// TIA Portal project "Lab6" (V16)

(* hardware
DEVICE "S71500/ET200MP station_1"  S7-1500 station
   slot 0: "Perfil soporte_0"  Rack  6ES7 590-1***0-0AA0
   slot 0: "PM 70W 120/230VAC"  PM 70W 120/230VAC  6EP1332-4BA00
   slot 1: "PLC_1"  CPU 1512C-1 PN  6ES7 512-1CK00-0AB0  V1.8
      slot 3: "Display de la CPU_1"  6ES7591-1AA00-0AA0
      slot 32768: "Interfaz PROFINET_1"  X1
   slot 2: "CP 1542-5_1"  CP 1542-5  6GK7 542-5FX00-0XE0  V1.0
DEVICE "PC-System_1"  SIMATIC PC station
   slot 0: "Estación PC SIMATIC"  Rail  SIMATIC PC-Station  V1.0
      slot 125: "Stationmanager"  Station_Manager  V6.0.4
   slot 1: "HMI_RT_1"  WinCC RT Advanced  6AV2 104-0xxxx-xxxx  16.0.0.0
      slot 33792: "Interfaz del equipo"  Host interface
   slot 2: "IE general_1"  IE General  IE_CP  V8.2.0
DEVICE "HMI_1"  KTP700 Basic PN
   slot 0: "HMI_1"  KTP700 Basic PN  6AV2 123-2GB03-0AX0  16.0.0.0
   slot 1: "HMI_RT_2"  KTP700 Basic PN  6AV2 123-2GB03-0AX0  16.0.0.0
   slot 5: "HMI_1.IE_CP_1"  PROFINET Interface  16.0.0.0
      slot 1: "Interfaz PROFINET_1"  PROFINET Interface
         slot 1: "Port_1"  Port
DEVICE "SINAMICS G_1"  Sinamics.Device
   slot 0: "	_0"  Rail  SinamicsG120SVecto
   slot 0: "accionamiento_1"  G120 CU250S-2 PN Vector  6SL3246-0BA22-1FA0  4.7.6
      slot 1: "Interfaz PROFINET"  MDD-SinamicsG120-P
   slot 3: "PM240-2 IP20"  PM240-2 IP20  6SL3210-1PB13-8ULx  -
DEVICE "S71500/ET200MP station_2"  S7-1500 station
   slot 0: "Perfil soporte_0"  Rack  6ES7 590-1***0-0AA0
   slot 1: "PLC_2"  CPU 1512C-1 PN  6ES7 512-1CK00-0AB0  V1.8
      slot 3: "Display de la CPU_1"  6ES7591-1AA00-0AA0
      slot 32768: "Interfaz PROFINET_1"  X1
   slot 2: "CP 1542-5_1"  CP 1542-5  6GK7 542-5FX00-0XE0  V1.0
*)

// ===== PLC "PLC_1"  CPU 1512C-1 PN =====

VAR_GLOBAL   // PLC tag table "Tabla de variables estándar"
   "Referencia(°C)" AT %MD14 : Real;
   "PT100" AT %IW20 : Int;
   "Bombillo" AT %Q4.7 : Bool;
   "Temperatura_Normal" AT %MD0 : Real;
   "Temperatura_Medida" AT %MD4 : Real;
   "Star" AT %M10.0 : Bool;
   "Stop" AT %M20.1 : Bool;
   "Paro" AT %M100.2 : Bool;
   "Servomotor" AT %Q16.1 : Bool;
   "Error" AT %MD104 : Real;
   "Alarma_Referencia_Alcanzada" AT %Q0.2 : Bool;
   "Encender_Variador" AT %M12.0 : Bool;
   "Stop_fisico" AT %I30.2 : Bool;
   "Parofisico" AT %I30.3 : Bool;
   "Star_Fisico" AT %I30.1 : Bool;
   "MoverDerecha" AT %M10.3 : Bool;
   "Pid_Sintonizado" AT %M8.0 : Bool;
   "Alarma_Alta" AT %Q16.3 : Bool;
   "Alarma_Baja" AT %Q16.4 : Bool;
   "Variador" AT %Q16.7 : Bool;
   "Ventilador" AT %Q16.6 : Bool;
   "Pid_Manual" AT %M8.1 : Bool;
   "Servosistema" AT %M8.2 : Bool;
   "Pid_Discreto" AT %M8.3 : Bool;
   "Control_Discreto" AT %MD22 : Real;
   "Control_Servo" AT %MD26 : Real;
   "Control_Servo(1)" AT %MD30 : Real;
   "Tag_1" AT %Q16.5 : Bool;
   "Error_Temperatura" AT %MD34 : Real;
END_VAR

DATA_BLOCK "Bloque_1_DB"   // DB4
{ S7_Optimized_Access := 'TRUE' }
VERSION : 0.1
// stored: InstanceOfName Bloque_1
"Bloque_1"
BEGIN
END_DATA_BLOCK

DATA_BLOCK "Base_de_Datos"   // DB5
{ S7_Optimized_Access := 'TRUE' }
VERSION : 0.1
BEGIN
END_DATA_BLOCK

// folder: System blocks/Program resources

DATA_BLOCK "IEC_Timer_0_DB"   // DB2
{ S7_Optimized_Access := 'TRUE' }
AUTHOR : Simatic
FAMILY : IEC
NAME : IEC_TMR
VERSION : 1.0
// stored: InstanceOfName IEC_TIMER
"IEC_TIMER"
BEGIN
END_DATA_BLOCK

DATA_BLOCK "IEC_Timer_0_DB_1"   // DB6
{ S7_Optimized_Access := 'TRUE' }
AUTHOR : Simatic
FAMILY : IEC
NAME : IEC_TMR
VERSION : 1.0
// stored: InstanceOfName IEC_TIMER
"IEC_TIMER"
BEGIN
END_DATA_BLOCK

DATA_BLOCK "IEC_Timer_0_DB_2"   // DB7
{ S7_Optimized_Access := 'TRUE' }
AUTHOR : Simatic
FAMILY : IEC
NAME : IEC_TMR
VERSION : 1.0
// stored: InstanceOfName IEC_TIMER
"IEC_TIMER"
BEGIN
END_DATA_BLOCK

// folder: (top level)

DATA_BLOCK "SpeedAxis_1"   // DB3, Motion_DB
{ S7_Optimized_Access := 'TRUE' }
AUTHOR : SIMATIC
FAMILY : MC_1500
VERSION : 2.0
// stored: InstanceOfName TO_SpeedAxis
"TO_SpeedAxis"
BEGIN
   DynamicLimits.MaxAcceleration := 1000.0;
   DynamicLimits.MaxDeceleration := 1000.0;
   DynamicLimits.MaxJerk := 20000.0;
   DynamicDefaults.Acceleration := 200.0;
   DynamicDefaults.Deceleration := 200.0;
   DynamicDefaults.Jerk := 4000.0;
   DynamicDefaults.EmergencyDeceleration := 1000.0;
   Actor.Interface.AddressIn := 256;
   Actor.Interface.AddressOut := 256;
END_DATA_BLOCK

FUNCTION_BLOCK "Bloque_1"   // FB1, FBD
{ S7_Optimized_Access := 'TRUE' }
VERSION : 0.1
   VAR
      MC_POWER_Instance : MC_POWER;
      MC_RESET_Instance : MC_RESET;
      MC_MOVEJOG_Instance : MC_MOVEJOG;
   END_VAR
BEGIN

REGION Network 1
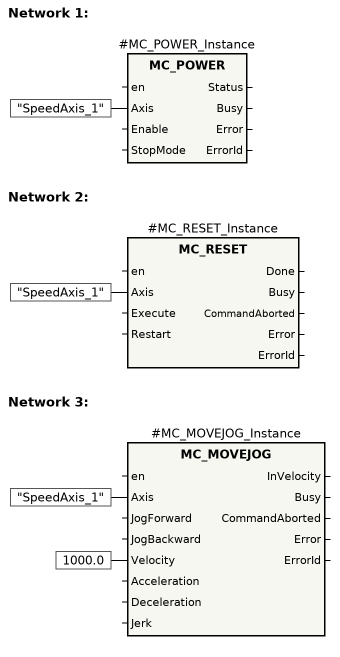
   #MC_POWER_Instance(Axis := "SpeedAxis_1");   // MC_POWER
END_REGION

REGION Network 2
   #MC_RESET_Instance(Axis := "SpeedAxis_1");   // MC_RESET
END_REGION

REGION Network 3
   #MC_MOVEJOG_Instance(Axis := "SpeedAxis_1", Velocity := 1000.0);   // MC_MOVEJOG
END_REGION
END_FUNCTION_BLOCK

ORGANIZATION_BLOCK "Main"   // OB1, LAD, ProgramCycle
TITLE = "Main Program Sweep (Cycle)"
{ S7_Optimized_Access := 'TRUE' }
VERSION : 0.1
   VAR_INPUT
      Initial_Call : Bool;   // Initial call of this OB
      Remanence : Bool;   // =True, if remanent data are available
   END_VAR
   VAR_TEMP
      Encender_Bombillo : Bool;
      Ventilador : Bool;
      calculo_error : Bool;
   END_VAR
BEGIN

REGION Network 1: Normalizar y escalar señal
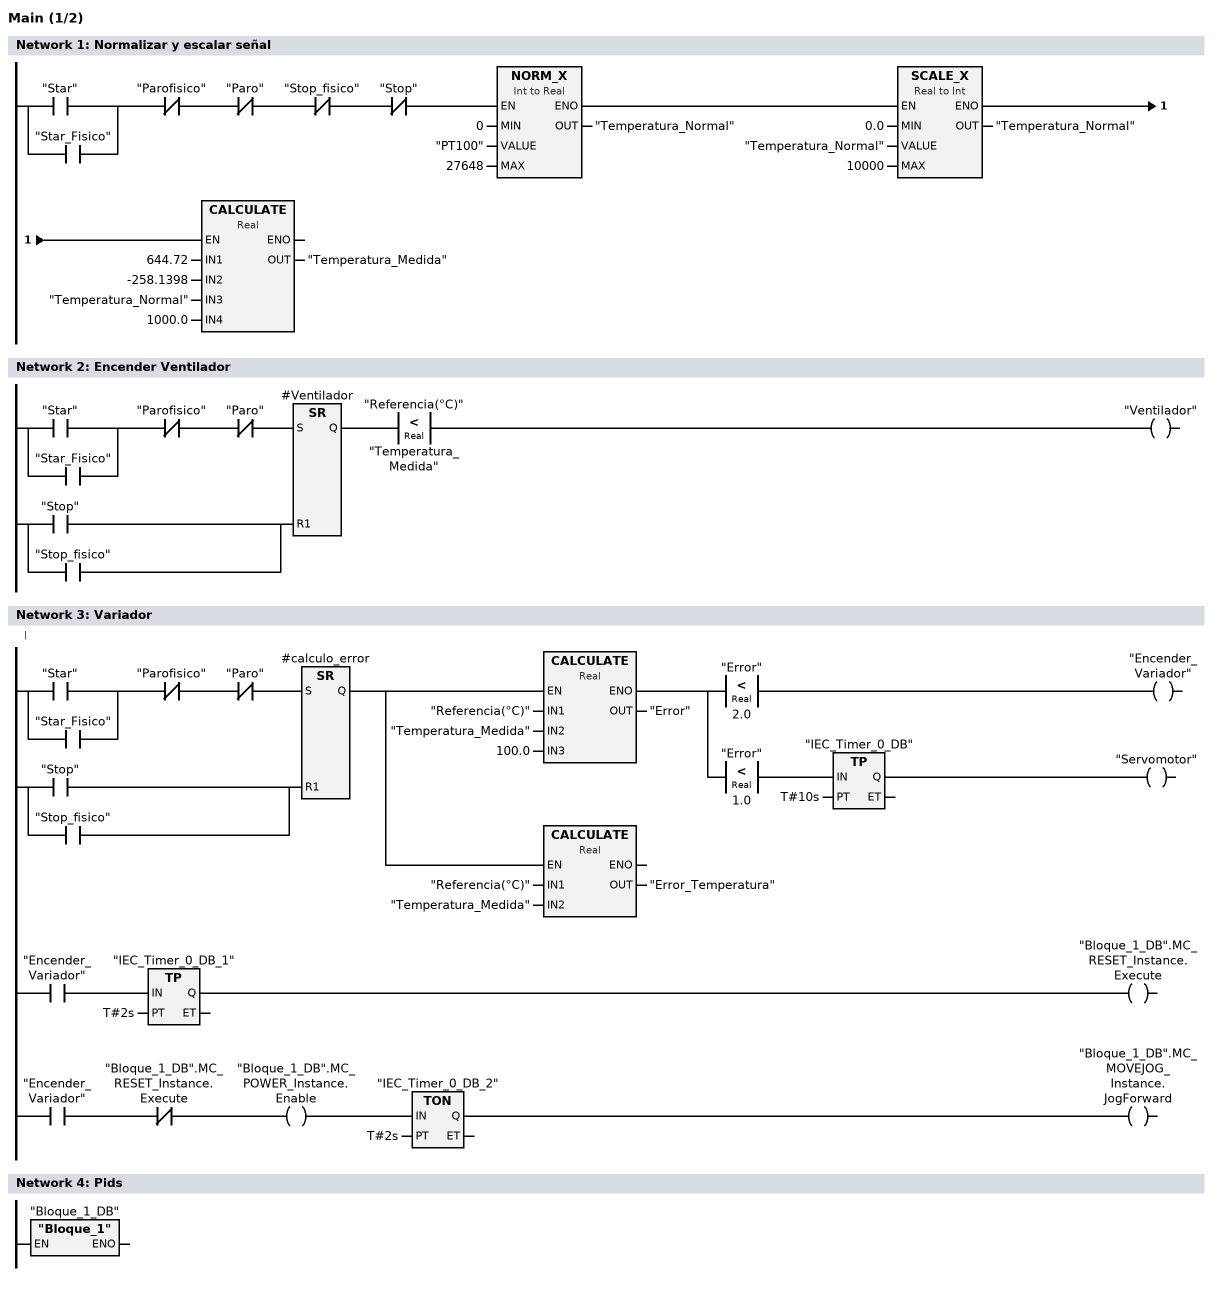
   RUNG wire#powerrail
      Contact( "Star" )
      wire#w1
      I_Contact( "Parofisico" )
      I_Contact( "Paro" )
      I_Contact( "Stop_fisico" )
      I_Contact( "Stop" )
      { S7_Templates := "[SrcType := Int, DestType := Real]" } Normalize(min := 0, value := "PT100", max := 27648, out => "Temperatura_Normal")
      { S7_Templates := "[SrcType := Real, DestType := Int]" } Scale(min := 0.0, value := "Temperatura_Normal", max := 10000, out => "Temperatura_Normal")
      { S7_Templates := "SrcType := Real"; S7_Expression := "(IN1*(IN3/IN4))+IN2" } Calculate(in1 := 644.72, in2 := -258.1398, in3 := "Temperatura_Normal", in4 := 1000.0, out => "Temperatura_Medida")
   END_RUNG
   RUNG wire#powerrail
      Contact( "Star_Fisico" )
   END_RUNG wire#w1
   // the same network as SCL:
   IF ("Star" OR "Star_Fisico") AND NOT "Parofisico" AND NOT "Paro" AND NOT "Stop_fisico" AND NOT "Stop" THEN
       "Temperatura_Normal" := NORM_X(MIN := 0, VALUE := "PT100", MAX := 27648);
       "Temperatura_Normal" := SCALE_X(MIN := 0.0, VALUE := "Temperatura_Normal", MAX := 10000);
       "Temperatura_Medida" := (644.72*("Temperatura_Normal"/1000.0))+(-258.1398);
   END_IF;
END_REGION

REGION Network 2: Encender Ventilador
   RUNG wire#powerrail
      Contact( "Star" )
      wire#w1
      I_Contact( "Parofisico" )
      I_Contact( "Paro" )
      S_SR(operand := #Ventilador, r1 := wire#w2)
      { S7_Templates := "SrcType := Real" } LT_Contact(in1 := "Referencia(°C)", in2 := "Temperatura_Medida")
      Coil( "Ventilador" )
   END_RUNG
   RUNG wire#powerrail
      Contact( "Star_Fisico" )
   END_RUNG wire#w1
   RUNG wire#powerrail
      Contact( "Stop" )
   END_RUNG wire#w2
   RUNG wire#powerrail
      Contact( "Stop_fisico" )
   END_RUNG wire#w2
   // the same network as SCL:
   IF ("Star" OR "Star_Fisico") AND NOT "Parofisico" AND NOT "Paro" THEN
       #Ventilador := TRUE;   // SR flip-flop
   END_IF;
   IF "Stop" OR "Stop_fisico" THEN #Ventilador := FALSE; END_IF;
   "Ventilador" := #Ventilador AND ("Referencia(°C)" < "Temperatura_Medida");
END_REGION

REGION Network 3: Variador
   // l
   IF ("Star" OR "Star_Fisico") AND NOT "Parofisico" AND NOT "Paro" THEN
       #calculo_error := TRUE;   // SR flip-flop
   END_IF;
   IF "Stop" OR "Stop_fisico" THEN #calculo_error := FALSE; END_IF;
   IF #calculo_error THEN
       "Error" := ABS(100.0*("Referencia(°C)"-"Temperatura_Medida")/("Referencia(°C)"));
   END_IF;
   "Encender_Variador" := #calculo_error AND ("Error" < 2.0);
   "IEC_Timer_0_DB".TP(IN := #calculo_error AND ("Error" < 1.0), PT := T#10s);
   "Servomotor" := "IEC_Timer_0_DB".Q;
   IF #calculo_error THEN "Error_Temperatura" := "Referencia(°C)"-"Temperatura_Medida"; END_IF;
   "IEC_Timer_0_DB_1".TP(IN := "Encender_Variador", PT := T#2s);
   "Bloque_1_DB".MC_RESET_Instance.Execute := "IEC_Timer_0_DB_1".Q;
   "Bloque_1_DB".MC_POWER_Instance.Enable := "Encender_Variador" AND NOT "Bloque_1_DB".MC_RESET_Instance.Execute;
   "IEC_Timer_0_DB_2".TON(IN := "Bloque_1_DB".MC_POWER_Instance.Enable, PT := T#2s);
   "Bloque_1_DB".MC_MOVEJOG_Instance.JogForward := "IEC_Timer_0_DB_2".Q;
END_REGION

REGION Network 4: Pids
   RUNG wire#powerrail
      "Bloque_1_DB"()
   END_RUNG
   // the same network as SCL:
   "Bloque_1_DB"();   // "Bloque_1"
END_REGION

REGION Network 5: Alarmas
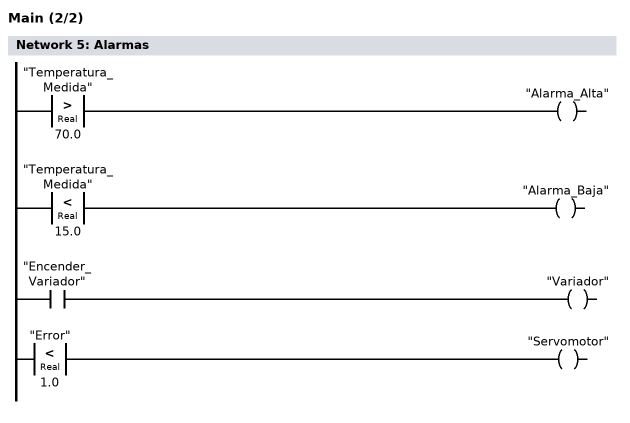
   RUNG wire#powerrail
      { S7_Templates := "SrcType := Real" } GT_Contact(in1 := "Temperatura_Medida", in2 := 70.0)
      Coil( "Alarma_Alta" )
   END_RUNG
   RUNG wire#powerrail
      { S7_Templates := "SrcType := Real" } LT_Contact(in1 := "Temperatura_Medida", in2 := 15.0)
      Coil( "Alarma_Baja" )
   END_RUNG
   RUNG wire#powerrail
      Contact( "Encender_Variador" )
      Coil( "Variador" )
   END_RUNG
   RUNG wire#powerrail
      { S7_Templates := "SrcType := Real" } LT_Contact(in1 := "Error", in2 := 1.0)
      Coil( "Servomotor" )
   END_RUNG
   // the same network as SCL:
   "Alarma_Alta" := "Temperatura_Medida" > 70.0;
   "Alarma_Baja" := "Temperatura_Medida" < 15.0;
   "Variador" := "Encender_Variador";
   "Servomotor" := "Error" < 1.0;
END_REGION
END_ORGANIZATION_BLOCK

ORGANIZATION_BLOCK "Cyclic interrupt_1"   // OB31, LAD, CyclicInterrupt
{ S7_Optimized_Access := 'TRUE' }
VERSION : 0.1
   VAR_INPUT
      Initial_Call : Bool;   // Initial call of this OB
      Event_Count : Int;   // Events discarded
   END_VAR
BEGIN

REGION Network 2: Sintonizado
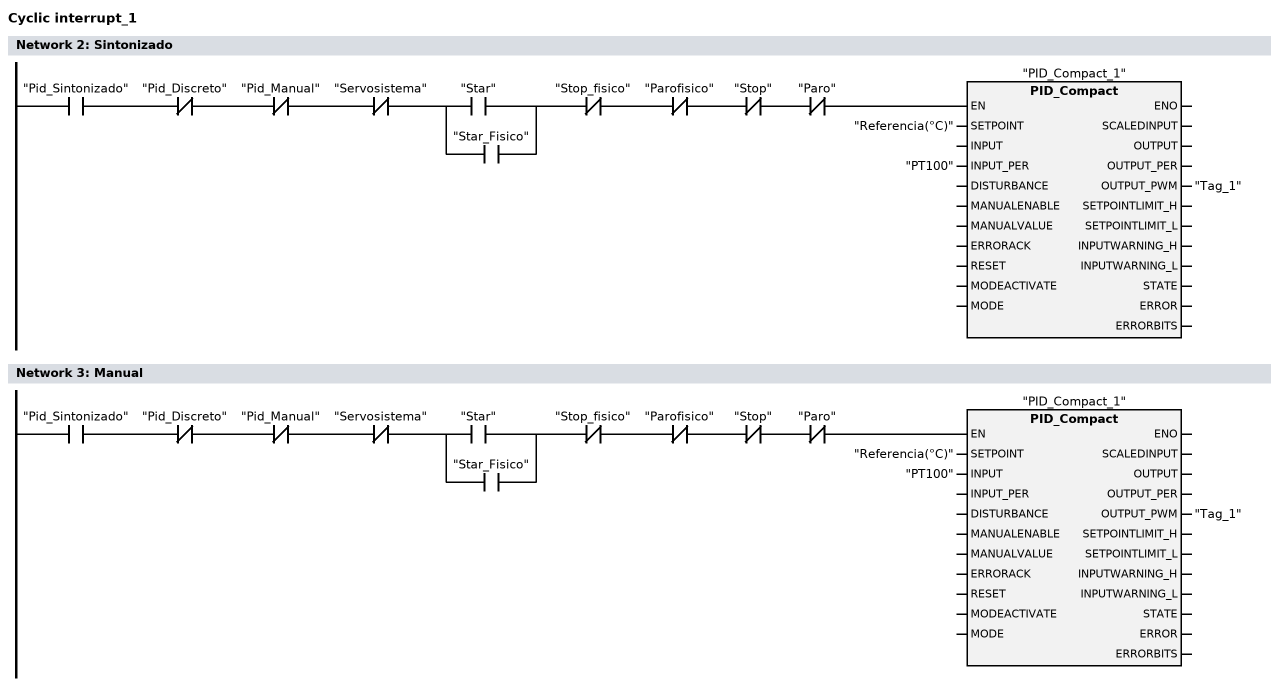
   IF "Pid_Sintonizado" AND NOT "Pid_Discreto" AND NOT "Pid_Manual" AND NOT "Servosistema" AND ("Star" OR "Star_Fisico") AND NOT "Stop_fisico" AND NOT "Parofisico" AND NOT "Stop" AND NOT "Paro" THEN
       "PID_Compact_1"(Setpoint := "Referencia(°C)", Input_PER := "PT100", Output_PWM => "Tag_1");   // PID_Compact
   END_IF;
END_REGION

REGION Network 3: Manual
   IF "Pid_Sintonizado" AND NOT "Pid_Discreto" AND NOT "Pid_Manual" AND NOT "Servosistema" AND ("Star" OR "Star_Fisico") AND NOT "Stop_fisico" AND NOT "Parofisico" AND NOT "Stop" AND NOT "Paro" THEN
       "PID_Compact_1"(Setpoint := "Referencia(°C)", Input := "PT100", Output_PWM => "Tag_1");   // PID_Compact
   END_IF;
END_REGION

REGION Network 4: Servosistema
END_REGION

REGION Network 5: Pid Discreto
END_REGION
END_ORGANIZATION_BLOCK

ORGANIZATION_BLOCK "Main_1"   // OB123, LAD, ProgramCycle
TITLE = "Main Program Sweep (Cycle)"
{ S7_Optimized_Access := 'TRUE' }
VERSION : 0.1
   VAR_INPUT
      Initial_Call : Bool;   // Initial call of this OB
      Remanence : Bool;   // =True, if remanent data are available
   END_VAR
BEGIN
END_ORGANIZATION_BLOCK

// ===== PLC "PLC_2"  CPU 1512C-1 PN =====

ORGANIZATION_BLOCK "Main"   // OB1, LAD, ProgramCycle
TITLE = "Main Program Sweep (Cycle)"
{ S7_Optimized_Access := 'TRUE' }
VERSION : 0.1
   VAR_INPUT
      Initial_Call : Bool;   // Initial call of this OB
      Remanence : Bool;   // =True, if remanent data are available
   END_VAR
BEGIN
END_ORGANIZATION_BLOCK

(* ===== HMI "HMI_RT_1" =====
system functions are stored by id; their names below are inferred from use
connection "HMI_Conexión_1": ETHERNET, S7_1500_OMS
connection "HMI_Conexión_4": ETHERNET, S7_1500_OMS

HMI tags "Tabla de variables estándar"
   "DatabaseName" : WString[254] AT %DB1.DBX0.0
   "ErrDesc" : WString[254], internal
   "TableName" : WString[254] AT %DB1.DBX0.0
   "Column1" : WString[254], internal
   "Column2" : WString[254], internal
   "Column3" : WString[254], internal
   "Referencia(°C)" : Real = PLC "Referencia(°C)" AT %MD14, 1 s
   "PT100" : Int = PLC PT100 AT %IW20, 1 s
   "Bombillo" : Bool = PLC Bombillo AT %Q4.7, 1 s
   "Temperatura_Normal" : Real = PLC Temperatura_Normal AT %MD0, 1 s
   "Temperatura_Medida" : Real = PLC Temperatura_Medida AT %MD4, 1 s
   "Star" : Bool = PLC Star AT %M10.0, 1 s
   "Stop" : Bool = PLC Stop AT %M20.1, 1 s
   "Paro" : Bool = PLC Paro AT %M100.2, 1 s
   "Servomotor" : Bool = PLC Servomotor AT %Q16.1, 1 s
   "Error" : Real = PLC Error AT %MD104, 1 s
   "Alarma_Referencia_Alcanzada" : Bool = PLC Alarma_Referencia_Alcanzada AT %Q0.2, 1 s
   "Encender_Variador" : Bool = PLC Encender_Variador AT %M12.0, 1 s
   "Stop_fisico" : Bool = PLC Stop_fisico AT %I30.2, 1 s
   "Parofisico" : Bool = PLC Parofisico AT %I30.3, 1 s
   "Star_Fisico" : Bool = PLC Star_Fisico AT %I30.1, 1 s
   "MoverDerecha" : Bool = PLC MoverDerecha AT %M10.3, 1 s
   "Pid_Sintonizado" : Bool = PLC Pid_Sintonizado AT %M8.0, 1 s
   "Alarma_Alta" : Bool = PLC Alarma_Alta AT %Q16.3, 1 s
   "Alarma_Baja" : Bool = PLC Alarma_Baja AT %Q16.4, 1 s
   "Variador" : Bool = PLC Variador AT %Q16.7, 1 s
   "Ventilador" : Bool = PLC Ventilador AT %Q16.6, 1 s
   "Pid_Manual" : Bool = PLC Pid_Manual AT %M8.1, 1 s
   "Servosistema" : Bool = PLC Servosistema AT %M8.2, 1 s
   "Pid_Discreto" : Bool = PLC Pid_Discreto AT %M8.3, 1 s
   "Tag_1" : Bool = PLC Tag_1 AT %Q16.5, 1 s
   "Error_Temperatura" : Real = PLC Error_Temperatura AT %MD34, 1 s

screen "Base de Datos" 800x600
   Button "Botón_1" at 22,16 size 209x32; TextOff 'Volver Panel de Control'
      on Press: function_efd93a16()
   IOField "Campo ES_1" at 217,133 size 109x32; FormatPattern 999.99999; Unit °C
      ProcessValue <- "Referencia(°C)"
   IOField "Campo ES_3" at 218,174 size 110x32; FormatPattern 999.99999; Unit °C
      ProcessValue <- "Error"
   TextField "Campo de texto_3" at 163,183 size 40x23; Text 'Error'
   TextField "Campo de texto_2" at 40,142 size 163x23; Text 'Temperatura_Deseada'
   TextField "Campo de texto_4" at 41,101 size 148x23; Text 'Temperatura_Actual'
   IOField "Campo ES_2" at 217,92 size 108x32; FormatPattern 999.99999; Unit °C
      ProcessValue <- "Temperatura_Medida"
   TextField "Campo de texto_1" at 40,62 size 166x23; Text 'Datos Tomados del plc'

screen "Control_Temperatura" 800x600
   Button "Botón_1" at 241,140 size 100x30; TextOff 'Star'
      on Click: SetBit("Star")
   Button "Botón_2" at 241,266 size 100x30; TextOff 'Stop'
      on Click: InvertBit("Stop")
   Button "Botón_3" at 241,202 size 100x30; TextOff 'Paro'
      on Click: InvertBit("Paro")
   IOField "Campo ES_4" at 38,40 size 96x32; FormatPattern 999.99999
      ProcessValue <- "Referencia(°C)"
   TextField "Campo de texto_1" at 7,7 size 209x28; Text 'Temperatura_Deseada'
   Bar "Barra_1" at 390,125 size 141x303; MinimumValue 0; MaximumValue 150
      ProcessValue <- "Temperatura_Medida"
   GraphicView "Visor de gráficos_4" at 25,221 size 161x242; Picture "Gráfico_6"
      Visibility <- "Tag_1"
   GraphicView "Visor de gráficos_3" at 25,221 size 161x242; Picture "Gráfico_7"
      Visibility <- "Tag_1"
   IOField "Campo ES_5" at 56,309 size 98x21; FormatPattern 999.99999
      ProcessValue <- "Temperatura_Medida"
   GraphicView "Visor de gráficos_1" at 162,354 size 95x102; Picture "Gráfico_9"
      Visibility <- "Tag_1"
   GraphicView "Visor de gráficos_2" at 162,354 size 95x102; Picture "Gráfico_9"
      Visibility <- "Tag_1"
   TextField "Campo de texto_4" at 36,163 size 186x28; Text 'Temperatura_Actual'
   Circle "Círculo_1" at 354,9 size 65x65
      Appearance <- "Servomotor"
   Circle "Círculo_2" at 440,8 size 65x65
      Appearance <- "Variador"
   Circle "Círculo_3" at 558,8 size 65x65
      Appearance <- "Alarma_Alta"
   TextField "Campo de texto_5" at 363,72 size 54x28; Text 'Servo'
   TextField "Campo de texto_6" at 437,72 size 79x28; Text 'Variador'
   TextField "Campo de texto_7" at 536,72 size 101x28; Text 'Temp_Alta'
   Circle "Círculo_4" at 680,6 size 65x65
      Appearance <- "Alarma_Baja"
   TextField "Campo de texto_8" at 667,70 size 106x28; Text 'Temp_Baja'
   Button "Botón_4" at 585,187 size 140x30; TextOff 'Pid_Sintonizado'
      on Press: InvertBit("Pid_Sintonizado")
      Appearance <- "Pid_Sintonizado"
   Button "Botón_7" at 30,83 size 140x30; TextOn 'Base de Datos'; TextOff 'Base de Datos'
      on Click: ActivateScreen("Base de Datos", 0)
      on Press: ActivateScreen("Base de Datos", 0)
   Button "Botón_8" at 585,129 size 140x30; TextOff 'Pid_Manual'
      on Press: InvertBit("Pid_Manual")
      Appearance <- "Pid_Manual"
   Button "Botón_9" at 585,237 size 140x30; TextOff 'Servosistema'
      on Press: InvertBit("Servosistema")
      Appearance <- "Servosistema"
   Button "Botón_10" at 585,287 size 140x30; TextOff 'Pid_Discreto'
      on Press: InvertBit("Pid_Discreto")
      Appearance <- "Pid_Discreto"
   Button "Botón_5" at 585,367 size 140x30; TextOn 'Base de Datos'; TextOff 'Graficas'
      on Click: ActivateScreen("Grafica", 0)
      on Press: ActivateScreen("Grafica", 0)

screen "Grafica" 800x600
   TrendView "Visor de curvas_1" at 21,9 size 769x388
   IOField "Campo ES_1" at 114,433 size 100x20; FormatPattern 999.99999
      ProcessValue <- "Referencia(°C)"
   IOField "Campo ES_3" at 288,433 size 100x20; FormatPattern 999.99999
      ProcessValue <- "Error_Temperatura"
   TextField "Campo de texto_3" at 325,405 size 40x23; Text 'Error'
   TextField "Campo de texto_2" at 89,407 size 163x23; Text 'Temperatura_Deseada'
   IOField "Campo ES_4" at 490,433 size 100x20; FormatPattern 999.99999
      ProcessValue <- "Temperatura_Medida"
   TextField "Campo de texto_1" at 453,403 size 144x23; Text 'Temperatura Actual'
   Button "Botón_1" at 647,421 size 138x32; TextOff 'Volver'
      on Press: function_efd93a16()

VB script "Crear_Base_De_Datos"
   Dim connect, record, DBName, ErrorDesc, SQLTable
   DBName = SmartTags("DatabaseName")
   On Error Resume Next
   
   Set connect = CreateObject("ADODB.Connection")
   Set record = CreateObject("ADODB.Recordset")
   
   connect.Open = "Provider=MSDASQL; DSN=" & Name_DSN & ";"
   
   If Err.Number <> 0 Then
   	
   ErrorDesc = Err.Description & " (" & Err.Number & ")"
   
   SmartTags("ErrDesc") = ErrorDesc
   
   Set connect = Nothing
   Exit Sub
   End If
   
   SQLTable = "CREATE DATABASE " & DBName
   Set record = connect.Execute(SQLTable)
   
   If Err.Number <> 0 Then
   ErrorDesc = Err.Description & " (" & Err.Number & ")"
   SmartTags("ErrDesc") = ErrorDesc
   Set connect = Nothing 
   End If 
   connect.close 
   Set connect = Nothing 
   Set record  = Nothing 

VB script "Crear_Tabla"
    Dim connect, record, DBName, TableName, SQLtable, ErrorDesc, Column1, Column2, Column3
   
       DBName = SmartTags("DatabaseName")
       TableName = SmartTags("TableName")
       Column1 = SmartTags("Column1")
       Column2 = SmartTags("Column2")
       Column3 = SmartTags("Column3")
   
       On Error Resume Next
   
       Set connect = CreateObject("ADODB.Connection")
       Set record = CreateObject("ADODB.Recordset")
   
       connect.Open "Provider=MSDASQL;Initial Catalog=" & DBName & ";DSN=" & Name_DSN & ";"
   
       If Err.Number <> 0 Then
           ErrorDesc = Err.Description & " (" & Err.Number & ")"
           SmartTags("ErrDesc") = ErrorDesc
           Set connect = Nothing
           Exit Sub
       End If
   
       SQLtable = "CREATE TABLE " & TableName & " (fecha_hora TIMESTAMP NOT NULL DEFAULT CURRENT_DATE(), " & Column1 & " FLOAT, " & Column2 & " FLOAT, " & Column3 & " FLOAT)"
       connect.Execute SQLtable
   
       If Err.Number <> 0 Then
           ErrorDesc = Err.Description & " (" & Err.Number & ")"
           SmartTags("ErrDesc") = ErrorDesc
           connect.Close
           Set connect = Nothing
           Exit Sub
       End If
   
       connect.Close
       Set connect = Nothing
       Set record = Nothing

VB script "Insertar_Data"
   	Dim connect,record, DBName, TableName, ErrorDesc, SQLinsert, value1, value2, value3
   	
   	DBName = SmartTags("DatabaseName")
   	TableName=SmartTags("TableName")
   	value1=SmartTags("Referencia(°C)")
   	value2=SmartTags("Temperatura_Medida")
   	value3=SmartTags("Error")
   	On Error Resume Next
   	Set connect = CreateObject("ADODB.Connection")
   	Set record = CreateObject("ADODB.Recordset")
   	connect.Open = "Provider=MSDASQL;Initial Catalog=" & DBName & ";DSN=" & Name_DSN & ";"
   	
   	If Err.Number <> 0 Then
   	ErrorDesc = Err.Description & " (" & Err.Number & ")"
   	SmartTags("ErrDesc") = ErrorDesc
   	Set connect = Nothing
   	Exit Sub
   	End If
   	SQLinsert= "INSERT INTO " & TableName & "(Referencia(°C),Temperatura_Medida,Error)"&"VALUES ('" & value1 & "','" & value2 & "','" & value3 & "')"
   	Set record = connect.Execute(SQLinsert)
   	If Err.Number <> 0 Then
   	ErrorDesc = Err.Description & " (" & Err.Number & ")"
   	SmartTags("ErrDesc") = ErrorDesc
   	Set connect = Nothing
   	Exit Sub
   	End If
   	connect.close 
   	Set connect = Nothing 
   	Set record  = Nothing 
   	
*)

(* ===== HMI "HMI_RT_2" =====
system functions are stored by id; their names below are inferred from use
connection "HMI_Conexión_2": ETHERNET, SMART_S7_1500_OMS
connection "HMI_Conexión_3": ETHERNET, SMART_S7_1500_OMS
connection "HMI_Conexión_5": ETHERNET, SMART_S7_1500_OMS

HMI tags "Tabla de variables estándar"
   "Column1" : WString[254], internal
   "Column2" : WString[254], internal
   "Column3" : WString[254], internal
   "DatabaseName" : WString[254] AT %DB1.DBX0.0
   "ErrDesc" : WString[254], internal
   "TableName" : WString[254] AT %DB1.DBX0.0
   "Referencia(°C)" : Real = PLC "Referencia(°C)" AT %MD14, 1 s
   "PT100" : Int = PLC PT100 AT %IW20, 1 s
   "Bombillo" : Bool = PLC Bombillo AT %Q4.7, 1 s
   "Temperatura_Normal" : Real = PLC Temperatura_Normal AT %MD0, 1 s
   "Temperatura_Medida" : Real = PLC Temperatura_Medida AT %MD4, 1 s
   "Star" : Bool = PLC Star AT %M10.0, 1 s
   "Stop" : Bool = PLC Stop AT %M20.1, 1 s
   "Paro" : Bool = PLC Paro AT %M100.2, 1 s
   "Servomotor" : Bool = PLC Servomotor AT %Q16.1, 1 s
   "Error" : Real = PLC Error AT %MD104, 1 s
   "Alarma_Referencia_Alcanzada" : Bool = PLC Alarma_Referencia_Alcanzada AT %Q0.2, 1 s
   "Encender_Variador" : Bool = PLC Encender_Variador AT %M12.0, 1 s
   "Stop_fisico" : Bool = PLC Stop_fisico AT %I30.2, 1 s
   "Parofisico" : Bool = PLC Parofisico AT %I30.3, 1 s
   "Star_Fisico" : Bool = PLC Star_Fisico AT %I30.1, 1 s
   "MoverDerecha" : Bool = PLC MoverDerecha AT %M10.3, 1 s
   "Pid_Sintonizado" : Bool = PLC Pid_Sintonizado AT %M8.0, 1 s
   "Alarma_Alta" : Bool = PLC Alarma_Alta AT %Q16.3, 1 s
   "Alarma_Baja" : Bool = PLC Alarma_Baja AT %Q16.4, 1 s
   "Variador" : Bool = PLC Variador AT %Q16.7, 1 s
   "Ventilador" : Bool = PLC Ventilador AT %Q16.6, 1 s
   "Pid_Manual" : Bool = PLC Pid_Manual AT %M8.1, 1 s
   "Servosistema" : Bool = PLC Servosistema AT %M8.2, 1 s
   "Pid_Discreto" : Bool = PLC Pid_Discreto AT %M8.3, 1 s
   "Tag_1" : Bool = PLC Tag_1 AT %Q16.5, 1 s
   "Error_Temperatura" : Real = PLC Error_Temperatura AT %MD34, 1 s

text list "Nombre_imagen_lista_texto": 1 'Imagen raíz'

screen "Control_Temperatura" 800x480
   Button "Botón_1" at 241,140 size 100x30; TextOff 'Empezar'
      on Click: SetBit("Star")
   Button "Botón_2" at 241,266 size 100x30; TextOff 'emergencia'
      on Click: InvertBit("Stop")
   Button "Botón_3" at 241,202 size 100x30; TextOff 'Paro'
      on Click: InvertBit("Paro")
   IOField "Campo ES_4" at 38,40 size 96x32; FormatPattern 999.99999
      ProcessValue <- "Referencia(°C)"
   TextField "Campo de texto_1" at 7,7 size 209x28; Text 'Temperatura_Deseada'
   GraphicView "Visor de gráficos_4" at 567,180 size 161x242; Picture "Gráfico_6"
      Visibility <- "Tag_1"
   GraphicView "Visor de gráficos_3" at 566,180 size 161x242; Picture "Gráfico_7"
      Visibility <- "Tag_1"
   IOField "Campo ES_5" at 599,264 size 98x21; FormatPattern 999.99999
      ProcessValue <- "Temperatura_Medida"
   GraphicView "Visor de gráficos_1" at 696,324 size 95x102; Picture "Gráfico_9"
      Visibility <- "Tag_1"
   GraphicView "Visor de gráficos_2" at 696,328 size 95x102; Picture "Gráfico_9"
      Visibility <- "Tag_1"
   TextField "Campo de texto_4" at 559,132 size 186x28; Text 'Temperatura_Actual'
   Circle "Círculo_1" at 354,9 size 65x65
      Appearance <- "Servomotor"
   Circle "Círculo_2" at 440,8 size 65x65
      Appearance <- "Variador"
   Circle "Círculo_3" at 558,8 size 65x65
      Appearance <- "Alarma_Alta"
   TextField "Campo de texto_5" at 363,72 size 54x28; Text 'Servo'
   TextField "Campo de texto_6" at 437,72 size 79x28; Text 'Variador'
   TextField "Campo de texto_7" at 536,72 size 101x28; Text 'Temp_Alta'
   Circle "Círculo_4" at 680,6 size 65x65
      Appearance <- "Alarma_Baja"
   TextField "Campo de texto_8" at 667,70 size 106x28; Text 'Temp_Baja'
   Button "Botón_4" at 9,193 size 140x30; TextOff 'Pid_Sintonizado'
      on Press: InvertBit("Pid_Sintonizado")
      Appearance <- "Pid_Sintonizado"
   Button "Botón_7" at 7,88 size 140x30; TextOff 'Base de Datos'
      on Click: ActivateScreen("Base de Datos", 0)
      on Press: ActivateScreen("Base de Datos", 0)
   Button "Botón_8" at 9,139 size 140x30; TextOff 'Pid_Manual'
      on Press: InvertBit("Pid_Manual")
      Appearance <- "Pid_Manual"
   Button "Botón_9" at 9,296 size 140x30; TextOff 'Servosistema'
      on Press: InvertBit("Servosistema")
      Appearance <- "Servosistema"
   Button "Botón_10" at 9,247 size 140x30; TextOff 'Pid_Discreto'
      on Press: InvertBit("Pid_Discreto")
      Appearance <- "Pid_Discreto"
   Button "Botón_5" at 74,376 size 140x30; TextOn 'Base de Datos'; TextOff 'Graficas'
      on Click: ActivateScreen("Grafica", 0)
      on Press: ActivateScreen("Grafica", 0)
   Bar "Barra_3" at 419,132 size 48x290; MinimumValue 0; MaximumValue 100
      ProcessValue <- "Temperatura_Medida"

screen "Base de Datos" 800x480
   Button "Botón_1" at 22,16 size 209x32; TextOff 'Volver Panel de Control'
      on Press: function_efd93a16()
   IOField "Campo ES_1" at 217,133 size 109x32; FormatPattern 999.99999; Unit °C
      ProcessValue <- "Referencia(°C)"
   IOField "Campo ES_3" at 218,174 size 110x32; FormatPattern 999.99999; Unit °C
      ProcessValue <- "Error"
   TextField "Campo de texto_3" at 163,183 size 40x23; Text 'Error'
   TextField "Campo de texto_2" at 40,142 size 163x23; Text 'Temperatura_Deseada'
   TextField "Campo de texto_4" at 41,101 size 148x23; Text 'Temperatura_Actual'
   IOField "Campo ES_2" at 217,92 size 108x32; FormatPattern 999.99999; Unit °C
      ProcessValue <- "Temperatura_Medida"
   TextField "Campo de texto_1" at 40,62 size 166x23; Text 'Datos Tomados del plc'

screen "Grafica" 800x480
   TrendView "Visor de curvas_1" at 21,9 size 769x388
   IOField "Campo ES_1" at 114,433 size 100x20; FormatPattern 999.99999
      ProcessValue <- "Referencia(°C)"
   IOField "Campo ES_3" at 288,433 size 100x20; FormatPattern 999.99999
      ProcessValue <- "Error_Temperatura"
   TextField "Campo de texto_3" at 325,405 size 40x23; Text 'Error'
   TextField "Campo de texto_2" at 89,407 size 163x23; Text 'Temperatura_Deseada'
   IOField "Campo ES_4" at 490,433 size 100x20; FormatPattern 999.99999
      ProcessValue <- "Temperatura_Medida"
   TextField "Campo de texto_1" at 453,403 size 144x23; Text 'Temperatura Actual'
   Button "Botón_1" at 647,421 size 138x32; TextOff 'Volver'
      on Press: function_efd93a16()
*)